SUBAPPLICATION Uebung_030 (* LED_PWM Blinkende LED *)
  (* Standard: 61499-2; Description: Copyright (c) 2023 Meisterschulen am Ostbahnhof This program and the accompanying materials are made available under the terms of the Eclipse Public License 2.0 which is available at https://www.eclipse.org/legal/epl-2.0/ SPDX-License-Identifier: EPL-2.0 *)
  (* Version 1.0, 2023-10-23, Franz Höpfinger, Meisterschulen am Ostbahnhof *)
  IMPORT logiBUS::io::DI::logiBUS_DI::Input_I1;
  IMPORT logiBUS::io::DI::logiBUS_DI::Input_I2;
  IMPORT logiBUS::io::DI::logiBUS_DI::Input_I3;
  IMPORT logiBUS::io::DI::logiBUS_DI::Input_I4;
  IMPORT logiBUS::io::DO_LED::LED_FREQ;
  IMPORT logiBUS::io::DQ::logiBUS_DO::Output_Q1;
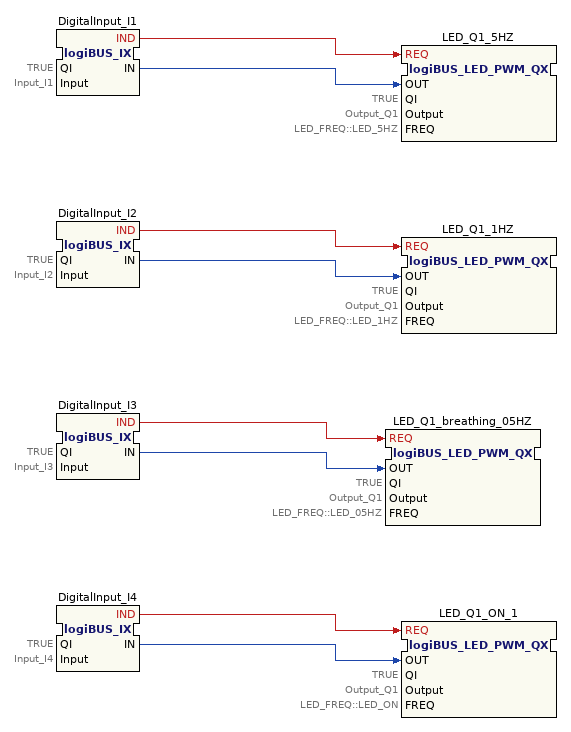
  FBS
    LED_Q1_5HZ : logiBUS::io::DO_LED::logiBUS_LED_PWM_QX(QI := TRUE, Output := Output_Q1, FREQ := LED_FREQ::LED_5HZ);
    DigitalInput_I1 : logiBUS::io::DI::logiBUS_IX(QI := TRUE, Input := Input_I1);
    LED_Q1_1HZ : logiBUS::io::DO_LED::logiBUS_LED_PWM_QX(QI := TRUE, Output := Output_Q1, FREQ := LED_FREQ::LED_1HZ);
    DigitalInput_I2 : logiBUS::io::DI::logiBUS_IX(QI := TRUE, Input := Input_I2);
    LED_Q1_breathing_05HZ : logiBUS::io::DO_LED::logiBUS_LED_PWM_QX(QI := TRUE, Output := Output_Q1, FREQ := LED_FREQ::LED_05HZ);
    DigitalInput_I3 : logiBUS::io::DI::logiBUS_IX(QI := TRUE, Input := Input_I3);
    DigitalInput_I4 : logiBUS::io::DI::logiBUS_IX(QI := TRUE, Input := Input_I4);
    LED_Q1_ON_1 : logiBUS::io::DO_LED::logiBUS_LED_PWM_QX(QI := TRUE, Output := Output_Q1, FREQ := LED_FREQ::LED_ON);
  END_FBS
  EVENT_CONNECTIONS
    DigitalInput_I1.IND TO LED_Q1_5HZ.REQ;
    DigitalInput_I2.IND TO LED_Q1_1HZ.REQ;
    DigitalInput_I3.IND TO LED_Q1_breathing_05HZ.REQ;
    DigitalInput_I4.IND TO LED_Q1_ON_1.REQ;
  END_CONNECTIONS
  DATA_CONNECTIONS
    DigitalInput_I1.IN TO LED_Q1_5HZ.OUT;
    DigitalInput_I2.IN TO LED_Q1_1HZ.OUT;
    DigitalInput_I3.IN TO LED_Q1_breathing_05HZ.OUT;
    DigitalInput_I4.IN TO LED_Q1_ON_1.OUT;
  END_CONNECTIONS
END_SUBAPPLICATION
